KUKA KRL data list: ALGEBRA.dat

&ACCESS RV1
&REL 1
DEFDAT ALGEBRA PUBLIC
   DECL GLOBAL CONST REAL EPS = 1E-09
   GLOBAL STRUC VECTOR3_T REAL X, Y, Z
   GLOBAL STRUC MATRIX3_T REAL M00, M01, M02, M10, M11, M12, M20, M21, M22
ENDDAT
